// TIA Portal project "定时器学习模拟（主轴，油泵）" (V15.1)

(* hardware
DEVICE "S7-1200 station_1"  S7-1200 Station
   slot 0: "Rack_0"  S7-1200 Rack  Rack  V1.0
   slot 1: "PLC_1"  CPU 1214C DC/DC/DC  6ES7 214-1AG40-0XB0  V4.2
*)

// ===== PLC "PLC_1"  CPU 1214C DC/DC/DC =====

VAR_GLOBAL   // PLC tag table "默认变量表"
   ""启动"" AT %I0.0 : Bool;
   ""停止"" AT %I0.1 : Bool;
   ""正转"" AT %I0.2 : Bool;
   ""反转"" AT %I0.3 : Bool;
   ""急停"" AT %I0.4 : Bool;
   ""主轴急停"" AT %I0.5 : Bool;
   ""油泵电机急停"" AT %I0.6 : Bool;
   ""主轴继电器"" AT %Q0.0 : Bool;
   ""油泵继电器"" AT %Q0.1 : Bool;
   ""主轴正转"" AT %Q0.2 : Bool;
   ""主轴反转"" AT %Q0.3 : Bool;
   ""系统运行指示灯"" AT %Q0.4 : Bool;
   ""系统停止指示灯"" AT %Q0.5 : Bool;
   ""主轴运行指示灯"" AT %Q0.6 : Bool;
   ""油泵运行指示灯"" AT %Q0.7 : Bool;
END_VAR